PROGRAM MAIN
VAR
	a:INT;
	b:INT;
	c:INT;
	add1:FB_ADD;
END_VAR

add1(in1:=a , in2:=b , out=>c );

END_PROGRAM

(* stored: Version 1.1.0.1, ProductVersion 3.1.4024.3
   POU MAIN: Id {b30f7bc4-5585-48ba-bc0b-09674d757870}, SpecialFunc None *)
